PROGRAM MAIN_ExternalTick
VAR
	fbSetRtMode : FB_SetRtMode;
	fbGetRtMode : FB_GetRtMode;
	
	state : INT := 0;	
	bStart : BOOL; 
	hint: STRING;
END_VAR

VAR_OUTPUT 
	value AT %Q* : UDINT;	
END_VAR


fbSetRtMode(bExecute:=FALSE);
fbGetRtMode(bExecute:=FALSE);

CASE state OF
	0:
		IF(bStart = TRUE) THEN 		
			state:= 1;
			value:=100; // steps to decrement as Cyclic 
		END_IF
	1:
		IF fbGetRtMode.bBusy = FALSE THEN  
			IF  fbGetRtMode.bError = FALSE  THEN
				IF fbGetRtMode.rtMode = E_RtMode.RtMode_Cyclic THEN
					state:=2; //if Cyclic start simulation = decremtn
					hint := '..cycling...'; 		
				ELSE
					fbGetRtMode(bExecute:= TRUE);
				END_IF
			ELSE	
				state:= 101;
			END_IF			
		END_IF
	2: 
		value:=value-1; //decrementing Cyclic (near realtime speed) 
		IF value = 0 THEN
			state := 3;
			fbSetRtMode(bExecute:= TRUE, rtMode:=E_RtMode.RtMode_Externaltick);	
			hint := '!!! WAITING FOR EXTERNAL TICKS !!!'; 		
		END_IF
	3:
		IF  fbSetRtMode.bBusy = FALSE THEN  
			IF fbSetRtMode.bError = FALSE THEN
				fbGetRtMode(bExecute:= TRUE);//querying RtMode  
				state := 4;
				value:=100; // Steps to decrement by External Ticks 						
			ELSE
				state := 101;
			END_IF  
		END_IF
	4:
		IF fbGetRtMode.bBusy = FALSE THEN  
			IF  fbGetRtMode.bError = FALSE  THEN
				IF fbGetRtMode.rtMode = E_RtMode.RtMode_Externaltick THEN
					state:=5; //if ExternalTick start decrementing by external ticks
				ELSE
					fbGetRtMode(bExecute:= TRUE);
				END_IF
			ELSE	
				state:= 102;
			END_IF			
		END_IF
	5: 
		value:=value-1; //decrementing as fast as possible 
		IF value = 0 THEN
			(*switch back to cyclic mode*)		
			fbSetRtMode(bExecute:= TRUE, rtMode:=E_RtMode.RtMode_Cyclic);
			state := 6;
		END_IF
	6:
		IF  fbSetRtMode.bBusy = FALSE THEN
			IF fbSetRtMode.bError = FALSE THEN
				hint := '..restart...'; 		
				state := 0;				
			ELSE
				state := 103;
			END_IF  
		END_IF	 	
END_CASE

END_PROGRAM

(* stored: Version 1.1.0.1, ProductVersion 3.1.4024.4
   POU MAIN_ExternalTick: Id {13441f1d-4eeb-4aed-abfe-d80e60f000dc}, SpecialFunc None *)
